PROGRAM Fridge3B
VAR
// Inputs (simulated)
	
	
	
	

	
	tDoorOpenThreshold : TIME := T#10S; //Time from door opening after which alarm turns on
	
	fbTimerDoorAlarm : TON;
	bAlarmLatched : BOOL; // Latched alaram state
END_VAR

// Light control (same as before)
GVL_Var.bLight := GVL_Var.bDoorOpen;
// Door alarm timer
fbTimerDoorAlarm(IN := GVL_Var.bDoorOpen, PT := tDoorOpenThreshold);
// Alarm logic with latching
IF fbTimerDoorAlarm.Q THEN
	bAlarmLatched := TRUE;
END_IF
// Reset alarm
IF GVL_Var.bAlarmReset THEN
	bAlarmLatched := FALSE;
END_IF
// Output alarm
GVL_Var.bAlarmOut := bAlarmLatched;
// Compressor control
IF GVL_Var.fTempActual > GVL_Var.fTempSet THEN
	GVL_Var.bCompressor := TRUE; // Warm: turn ON
ELSE
	GVL_Var.bCompressor := FALSE; // Cold: turn OFF
END_IF

END_PROGRAM

(* stored: Version 1.1.0.1, ProductVersion 3.1.4026.18
   POU Fridge3B: Id {ac3873f4-0ded-4787-9709-7e71ea45fcf7}, SpecialFunc None *)
